FUNCTION_BLOCK ABSTRACT FB_AbstractDevice IMPLEMENTS I_Device

VAR
	_name : STRING;
END_VAR

PROPERTY name : STRING
GET
name : _name;
END_GET
SET
_name := name;
END_SET
END_PROPERTY

END_FUNCTION_BLOCK

(* stored: Version 1.1.0.1
   POU FB_AbstractDevice: Id {4e4396b5-d1e6-4aba-b839-c73d5780e046}, SpecialFunc None
   Property name: Id {76877351-33b9-484e-a926-f6dbe89aa53f}
   Get Get: Id {a4e1970a-7137-479b-80e2-527455a01b95}
   Set Set: Id {594844e5-4337-45d2-a5ed-fd2ce7ee4a0f} *)
